// TIA Portal V15.1 export
// export: Created 2020-06-12T07:35:53.8974609Z, ExportSetting None, DisplayName Totally Integrated Automation Portal, DisplayVersion V15.1, DisplayName TIA Portal Openness, DisplayVersion V15.1, DisplayName STEP 7 Professional, DisplayVersion V15.1, DisplayName STEP 7 Safety, DisplayVersion V15.1, DisplayName WinCC Advanced, DisplayVersion V15.1
FUNCTION "RCW_PTCtrl" : Void   // FC153, FBD
TITLE = RCW: pumps speed controler
{ S7_Optimized_Access := 'TRUE' }
// stored: SetENOAutomatically False
   VAR_TEMP
      tSpdMax : Real;
      tSpdAdd : Real;
      tRelativeFlow : Real;
      tSumFlow : Real;
      tContLocked : Bool;
      tContOut : Real;
      tContIsOn : Bool;
      tFanSpeedMin : Real;
      tFanSpeedMax : Real;
   END_VAR
BEGIN

REGION Network 1: TODO
END_REGION

REGION Network 2: Pressure controller
   // !! WARNING: This is NOT controller call. See a blocks 'ContrFast_call'
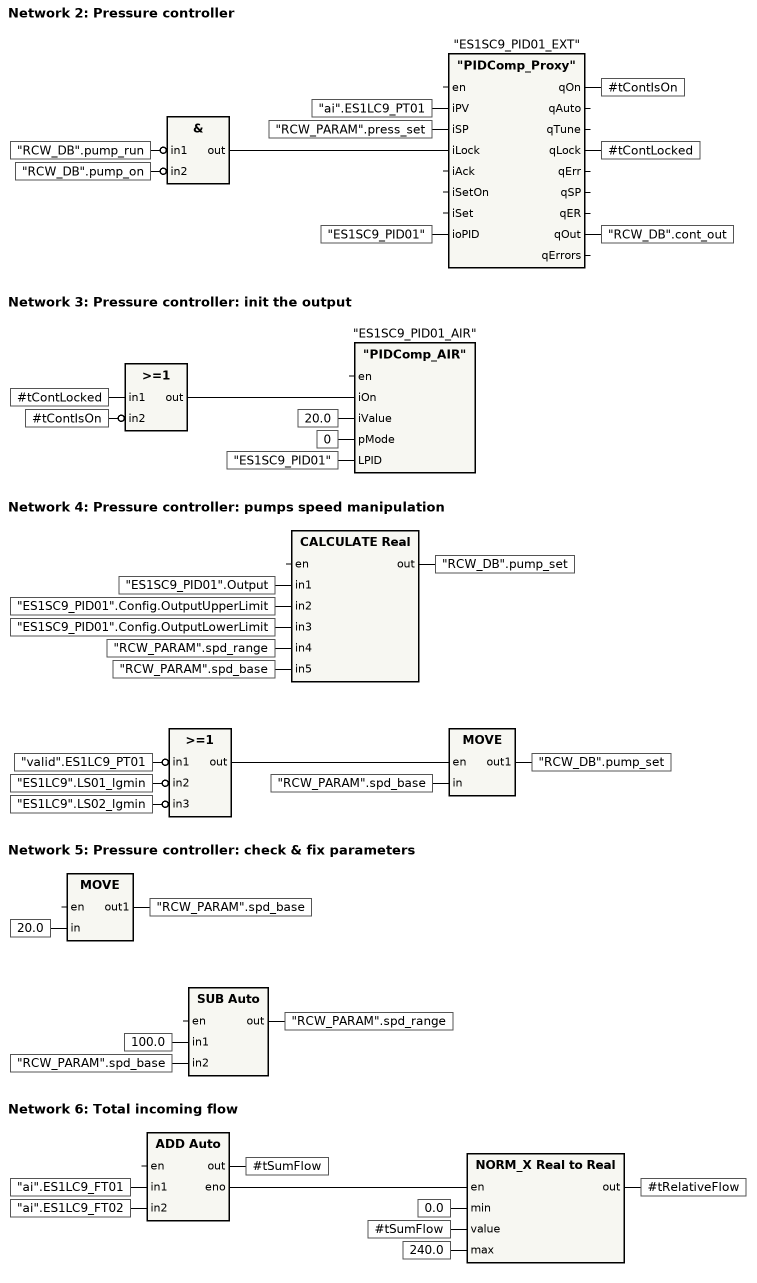
   "ES1SC9_PID01_EXT"(iPV := "ai".ES1LC9_PT01,   // "PIDComp_Proxy"
                      iSP := "RCW_PARAM".press_set,
                      iLock := NOT "RCW_DB".pump_run AND NOT "RCW_DB".pump_on,
                      ioPID := "ES1SC9_PID01",
                      qOn => #tContIsOn,
                      qLock => #tContLocked,
                      qOut => "RCW_DB".cont_out);
END_REGION

REGION Network 3: Pressure controller: init the output
   "ES1SC9_PID01_AIR"(iOn := #tContLocked OR NOT #tContIsOn, iValue := 20.0, pMode := 0, LPID := "ES1SC9_PID01");   // "PIDComp_AIR"
END_REGION

REGION Network 4: Pressure controller: pumps speed manipulation
   "RCW_DB".pump_set := (("ES1SC9_PID01".Output - "ES1SC9_PID01".Config.OutputLowerLimit) / ("ES1SC9_PID01".Config.OutputUpperLimit - "ES1SC9_PID01".Config.OutputLowerLimit))*"RCW_PARAM".spd_range + "RCW_PARAM".spd_base;
   IF NOT "valid".ES1LC9_PT01 OR NOT "ES1LC9".LS01_lgmin OR NOT "ES1LC9".LS02_lgmin THEN
       "RCW_DB".pump_set := "RCW_PARAM".spd_base;
   END_IF;
END_REGION

REGION Network 5: Pressure controller: check & fix parameters
   "RCW_PARAM".spd_base := 20.0;
   "RCW_PARAM".spd_range := 100.0 - "RCW_PARAM".spd_base;
END_REGION

REGION Network 6: Total incoming flow
   #tSumFlow := "ai".ES1LC9_FT01 + "ai".ES1LC9_FT02;
   #tRelativeFlow := NORM_X(MIN := 0.0, VALUE := #tSumFlow, MAX := 240.0);
END_REGION

REGION Network 7: Temperature controller
   // !! WARNING: This is NOT controller call. See a blocks 'ContrSlow_call'
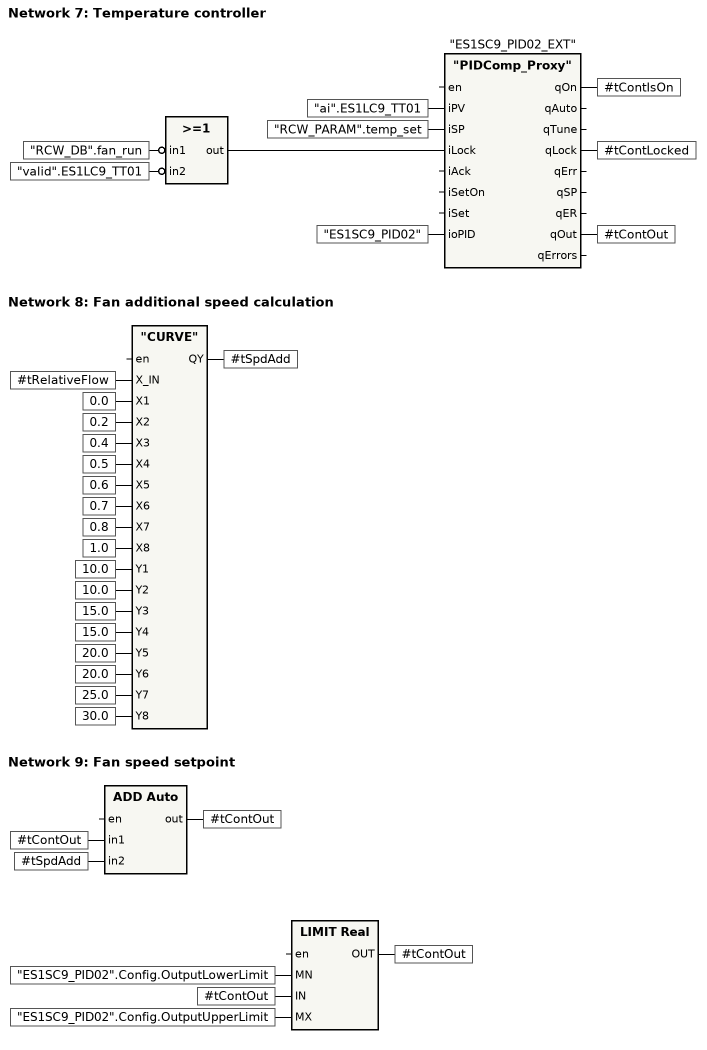
   "ES1SC9_PID02_EXT"(iPV := "ai".ES1LC9_TT01,   // "PIDComp_Proxy"
                      iSP := "RCW_PARAM".temp_set,
                      iLock := NOT "RCW_DB".fan_run OR NOT "valid".ES1LC9_TT01,
                      ioPID := "ES1SC9_PID02",
                      qOn => #tContIsOn,
                      qLock => #tContLocked,
                      qOut => #tContOut);
END_REGION

REGION Network 8: Fan additional speed calculation
   // Feedforward
   "CURVE"(X_IN := #tRelativeFlow,
           X1 := 0.0,
           X2 := 0.2,
           X3 := 0.4,
           X4 := 0.5,
           X5 := 0.6,
           X6 := 0.7,
           X7 := 0.8,
           X8 := 1.0,
           Y1 := 10.0,
           Y2 := 10.0,
           Y3 := 15.0,
           Y4 := 15.0,
           Y5 := 20.0,
           Y6 := 20.0,
           Y7 := 25.0,
           Y8 := 30.0,
           QY => #tSpdAdd);
END_REGION

REGION Network 9: Fan speed setpoint
   #tContOut := #tContOut + #tSpdAdd;
   #tContOut := LIMIT(MN := "ES1SC9_PID02".Config.OutputLowerLimit, IN := #tContOut, MX := "ES1SC9_PID02".Config.OutputUpperLimit);
END_REGION

REGION Network 10: AX1LD3.M01: Fan speed scaling
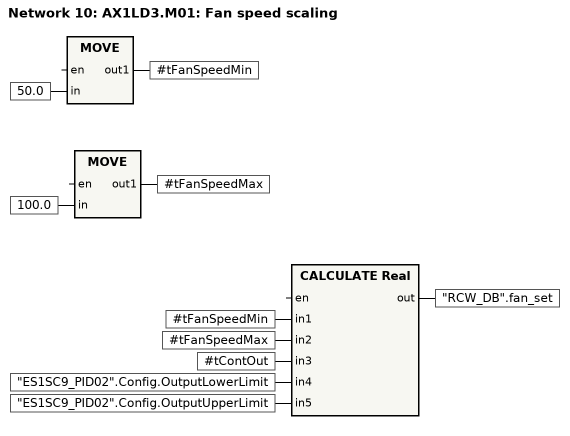
   #tFanSpeedMin := 50.0;
   #tFanSpeedMax := 100.0;
   "RCW_DB".fan_set := #tFanSpeedMin + (#tFanSpeedMax - #tFanSpeedMin) * ((#tContOut - "ES1SC9_PID02".Config.OutputLowerLimit) / ("ES1SC9_PID02".Config.OutputUpperLimit - "ES1SC9_PID02".Config.OutputLowerLimit));
END_REGION
END_FUNCTION
